// TIA Portal V17 export
// export: Created 2024-08-29T18:23:44.9716387Z, ExportSetting WithDefaults, DisplayName Totally Integrated Automation Portal, DisplayVersion V17 Update 7, DisplayName TIA Portal Openness, DisplayVersion V17 Update 7, DisplayName TIA Portal Version Control Interface, DisplayVersion V17, DisplayName SINAMICS Startdrive Advanced, DisplayVersion V17 SP2, DisplayName SINAMICS Startdrive G110M, G120, G120C, G120D, G120P, G115D, DisplayVersion V17 SP2, DisplayName SINAMICS Startdrive G130, G150, S120, S150, SINAMICS MV, S210, DisplayVersion V17 SP2, DisplayName STEP 7 Professional, DisplayVersion V17 Update 7, DisplayName STEP 7 Safety, DisplayVersion V17 Update 6, DisplayName WinCC Advanced / Unified PC, DisplayVersion V17 Update 7
FUNCTION "FC_CONTROL_PRINTER" : Void   // FC325, LAD
{ S7_Optimized_Access := 'TRUE' }
VERSION : 0.1
// stored: AutoNumber false, IsIECCheckEnabled false, SetENOAutomatically false, UDAEnableTagReadback false
BEGIN

REGION Network 1
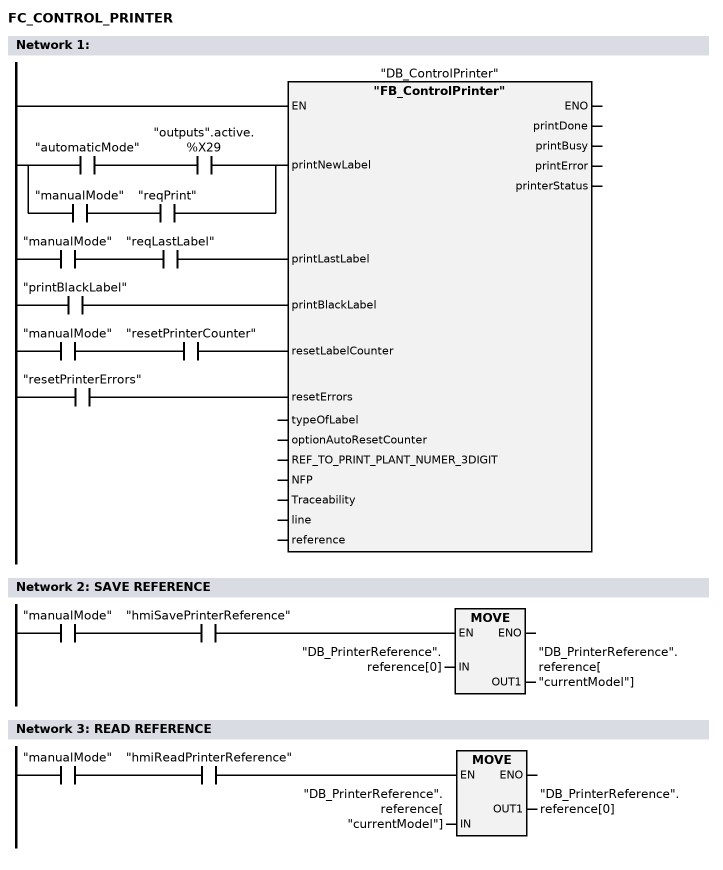
   RUNG wire#powerrail
      "DB_ControlPrinter"(printNewLabel := wire#w1, printLastLabel := wire#w2, printBlackLabel := wire#w3, resetLabelCounter := wire#w4, resetErrors := wire#w5, typeOfLabel :=, optionAutoResetCounter :=, REF_TO_PRINT_PLANT_NUMER_3DIGIT :=, NFP :=, Traceability :=, line :=, reference :=, printDone =>, printBusy =>, printError =>, printerStatus =>)
   END_RUNG
   RUNG wire#powerrail
      Contact( "automaticMode" )
      Contact( "outputs".active.%X29 )
   END_RUNG wire#w1
   RUNG wire#powerrail
      Contact( "manualMode" )
      Contact( "reqPrint" )
   END_RUNG wire#w1
   RUNG wire#powerrail
      Contact( "manualMode" )
      Contact( "reqLastLabel" )
   END_RUNG wire#w2
   RUNG wire#powerrail
      Contact( "printBlackLabel" )
   END_RUNG wire#w3
   RUNG wire#powerrail
      Contact( "manualMode" )
      Contact( "resetPrinterCounter" )
   END_RUNG wire#w4
   RUNG wire#powerrail
      Contact( "resetPrinterErrors" )
   END_RUNG wire#w5
   // the same network as SCL:
   "DB_ControlPrinter"(printNewLabel := ("automaticMode" AND "outputs".active.%X29) OR ("manualMode" AND "reqPrint"),   // "FB_ControlPrinter"
                       printLastLabel := "manualMode" AND "reqLastLabel",
                       printBlackLabel := "printBlackLabel",
                       resetLabelCounter := "manualMode" AND "resetPrinterCounter",
                       resetErrors := "resetPrinterErrors");
END_REGION

REGION Network 2: SAVE REFERENCE
   RUNG wire#powerrail
      Contact( "manualMode" )
      Contact( "hmiSavePrinterReference" )
      Move(in := "DB_PrinterReference".reference[0], out1 => "DB_PrinterReference".reference["currentModel"])
   END_RUNG
   // the same network as SCL:
   IF "manualMode" AND "hmiSavePrinterReference" THEN
       "DB_PrinterReference".reference["currentModel"] := "DB_PrinterReference".reference[0];
   END_IF;
END_REGION

REGION Network 3: READ REFERENCE
   RUNG wire#powerrail
      Contact( "manualMode" )
      Contact( "hmiReadPrinterReference" )
      Move(in := "DB_PrinterReference".reference["currentModel"], out1 => "DB_PrinterReference".reference[0])
   END_RUNG
   // the same network as SCL:
   IF "manualMode" AND "hmiReadPrinterReference" THEN
       "DB_PrinterReference".reference[0] := "DB_PrinterReference".reference["currentModel"];
   END_IF;
END_REGION
END_FUNCTION
